FUNCTION_BLOCK fbAxisControl
VAR_IN_OUT
	Axis: ST_Axis;
END_VAR
VAR
	mcPower: MC_Power;
	mcReset: MC_Reset;
	mcHalt: MC_Halt;
	mcMoveAbs: MC_MoveAbsolute;
	mcMoveRel: MC_MoveRelative;
END_VAR

(* Update axis status *)
Axis.Axis();

(* Error and Reset transition overrides *)
IF mcReset.Done THEN
    Axis.State := E_AxisState.INIT;
ELSIF Axis.Axis.Status.Error THEN
    Axis.LastError := Axis.Axis.Status.ErrorId;
	Axis.State := E_AxisState.ERROR;
ELSIF mcPower.Error THEN
	Axis.LastError := mcPower.ErrorId;
	Axis.State := E_AxisState.ERROR;
ELSIF mcReset.Error THEN
	Axis.LastError := mcReset.ErrorId;
	Axis.State := E_AxisState.ERROR;
END_IF;


(* Process other state changes *)
CASE Axis.State OF
	
    E_AxisState.INIT :
	Axis.DoReset := FALSE;
	Axis.DoHalt := FALSE;
	Axis.DoMoveAbs := FALSE;
	Axis.DoMoveRel := FALSE;
	Axis.Error := FALSE;
	Axis.LastError := 0;
	Axis.State := E_AxisState.READY;


	E_AxisState.READY :
	IF Axis.Axis.NcToPlc.StateDWord.8 (* HasJob *) THEN
		Axis.State := E_AxisState.BUSY;
    ELSIF mcReset.Busy OR mcHalt.Busy OR mcMoveAbs.Busy OR mcMoveRel.Busy THEN
		Axis.State := E_AxisState.BUSY;
	ELSIF Axis.DoMoveAbs THEN
		mcMoveAbs.Execute := TRUE;
		Axis.State := E_AxisState.BUSY;
	ELSIF Axis.DoMoveRel THEN
		mcMoveRel.Execute := TRUE;
		Axis.State := E_AxisState.BUSY;
	END_IF;

	
	E_AxisState.BUSY :
	(* Move Absolute *)
	Axis.DoMoveAbs := FALSE;
	IF mcMoveAbs.Execute AND NOT mcMoveAbs.Busy THEN
		IF mcMoveAbs.Error THEN
			Axis.LastError := mcMoveAbs.ErrorID;
		ELSIF mcMoveAbs.CommandAborted THEN
			Axis.LastError := 9999;
		ELSIF mcMoveAbs.Done THEN
			Axis.LastError := 0;
		END_IF;
		mcMoveAbs.Execute := FALSE;
	END_IF

	(* Move Relative *)
	Axis.DoMoveRel := FALSE;
	IF mcMoveRel.Execute AND NOT mcMoveRel.Busy THEN
		IF mcMoveRel.Error THEN
			Axis.LastError := mcMoveRel.ErrorID;
		ELSIF mcMoveRel.CommandAborted THEN
			Axis.LastError := 9999;
		ELSIF mcMoveRel.Done THEN
			Axis.LastError := 0;
		END_IF;
		mcMoveRel.Execute := FALSE;
	END_IF

	IF NOT (Axis.Axis.NcToPlc.StateDWord.8 (* HasJob *) OR mcReset.Busy OR mcHalt.Busy OR mcMoveAbs.Busy OR mcMoveRel.Busy) THEN
		Axis.State := E_AxisState.READY;
	END_IF;

	
	E_AxisState.ERROR :
	Axis.Error := TRUE;
	Axis.DoMoveAbs := FALSE;
	Axis.DoMoveRel := FALSE;

END_CASE


(* Execute mothion control function blocks. *)
ActPower();
ActMoveAbs();
ActMoveRel();
ActHalt();
ActReset();

(* Update Axis Status. *)
Axis.Status := Axis.Axis.Status;

ACTION ActHalt:
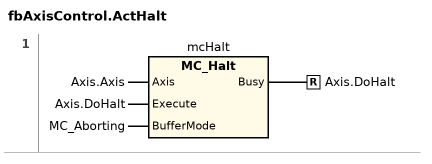
// NETWORK 1
mcHalt(Axis := Axis.Axis, Execute := Axis.DoHalt, BufferMode := MC_Aborting); // MC_Halt
Axis.DoHalt R= mcHalt.Busy;
END_ACTION

ACTION ActMoveAbs:
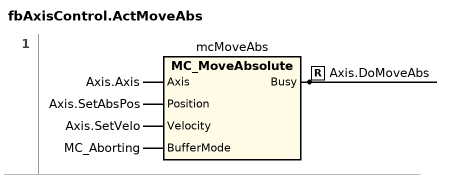
// NETWORK 1
mcMoveAbs(Axis := Axis.Axis, Position := Axis.SetAbsPos, Velocity := Axis.SetVelo, BufferMode := MC_Aborting); // MC_MoveAbsolute
Axis.DoMoveAbs R= mcMoveAbs.Busy;
END_ACTION

ACTION ActMoveRel:
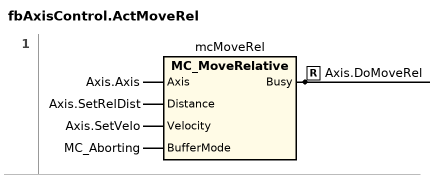
// NETWORK 1
mcMoveRel(
    Axis := Axis.Axis,
    Distance := Axis.SetRelDist,
    Velocity := Axis.SetVelo,
    BufferMode := MC_Aborting); // MC_MoveRelative
Axis.DoMoveRel R= mcMoveRel.Busy;
END_ACTION

ACTION ActPower:
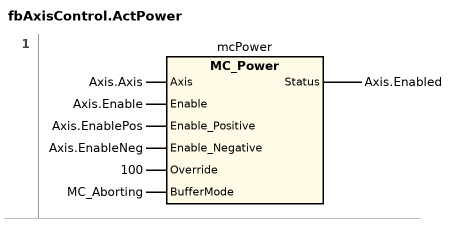
// NETWORK 1
mcPower(
    Axis := Axis.Axis,
    Enable := Axis.Enable,
    Enable_Positive := Axis.EnablePos,
    Enable_Negative := Axis.EnableNeg,
    Override := 100,
    BufferMode := MC_Aborting); // MC_Power
Axis.Enabled := mcPower.Status;
END_ACTION

ACTION ActReset:
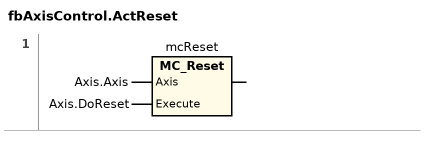
// NETWORK 1
mcReset(Axis := Axis.Axis, Execute := Axis.DoReset); // MC_Reset
END_ACTION

END_FUNCTION_BLOCK

(* stored: Version 1.1.0.1, ProductVersion 3.1.4020.12
   POU fbAxisControl: Id {db383e0a-e38c-4edf-93cc-4185104820fb}, SpecialFunc None
   Action ActHalt: Id {5b283866-d41c-462e-b67e-938a3f29984e}
   Action ActMoveAbs: Id {386f6c69-352c-47b0-8c47-bb0b008e1ce9}
   Action ActMoveRel: Id {39d79d3d-d4e8-4dd6-b153-cb87a727b7fe}
   Action ActPower: Id {b54c6d3d-b79c-4f5c-ab24-3c3f2108c000}
   Action ActReset: Id {48ae7dd0-e662-4220-915c-f299cce1e8d7} *)
